FUNCTION_BLOCK MY_XYZ_J (* Compute X^2-Y^2 in Java *)
  (* Standard: 61499-1 *)
  (* Version 0.2, 2011-08-21, JHC, Holobloc Inc, Moved algorithm text to a CDATA section. *)
  (* Version 0.1, 2006-09-06, JHC, Holobloc Inc, Made a SimpleFB. *)
  (* Version 0.0, 2001-10-09, JHC, Rockwell Automation *)
  (* Compiler header: package fb.rt.student; import fb.rt.math.*; *)
  (* Compiler Java IBM Jikes 1.0.6 *)
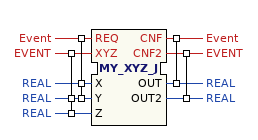
  EVENT_INPUT
    REQ WITH X, Y;
    XYZ : EVENT WITH Y, Z;
  END_EVENT
  EVENT_OUTPUT
    CNF WITH OUT;
    CNF2 : EVENT WITH OUT2;
  END_EVENT
  VAR_INPUT
    X : REAL;
    Y : REAL;
    Z : REAL;
  END_VAR
  VAR_OUTPUT
    OUT : REAL;
    OUT2 : REAL;
  END_VAR
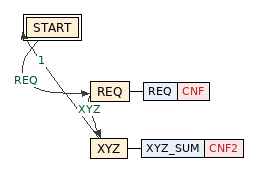
  EC_STATES
    START;
    REQ : REQ -> CNF;
    XYZ : XYZ_SUM -> CNF2;
  END_STATES
  EC_TRANSITIONS
    START TO REQ := REQ;
    REQ TO XYZ := XYZ;
    XYZ TO START := 1;
  END_TRANSITIONS
  ALGORITHM REQ IN Java:
OUT.value = (X.value+Y.value);
  END_ALGORITHM
  ALGORITHM XYZ_SUM IN Java:
OUT2.value = X.value + Y.value + Z.value;
  END_ALGORITHM
END_FUNCTION_BLOCK
